{attribute 'linkalways'} 
{attribute 'no_explicit_call' := 'This FB is a CLASS and must be accessed using methods or properties'}
{attribute 'enable_dynamic_creation'}
FUNCTION_BLOCK ChunkableServerResponse IMPLEMENTS I_ServerResponse
VAR
	serverResponse : I_ServerResponse;
	chunkedResponseManager : I_ChunkedResponseManager;
END_VAR

METHOD PUBLIC Accepted
VAR_INPUT
END_VAR
serverResponse.Accepted();
END_METHOD

METHOD PUBLIC Busy
VAR_INPUT
END_VAR
serverResponse.Busy();
END_METHOD

METHOD PUBLIC Error
VAR_INPUT
	Message : T_MAXSTRING;
END_VAR
serverResponse.Error(Message);
END_METHOD

METHOD FB_init : BOOL
VAR_INPUT
	bInitRetains : BOOL; // if TRUE, the retain variables are initialized (warm start / cold start)
	bInCopyCode : BOOL;  // if TRUE, the instance afterwards gets moved into the copy code (online change)
	ServerResponse : I_ServerResponse;
	ChunkedResponseManager : I_ChunkedResponseManager;
END_VAR
THIS^.serverResponse := ServerResponse;
This^.chunkedResponseManager := ChunkedResponseManager;
END_METHOD

PROPERTY PUBLIC Header : I_ServerResponseHeader
GET
Header := serverResponse.Header;
END_GET
END_PROPERTY

PROPERTY PUBLIC HeadersSent : BOOL
GET
HeadersSent := serverResponse.HeadersSent;
END_GET
END_PROPERTY

METHOD PUBLIC Pending
VAR_INPUT
	ResponseId : T_MAXSTRING;
	RetryDelayInMs : UDINT;
END_VAR
serverResponse.Pending(ResponseId, RetryDelayInMs);
END_METHOD

METHOD PUBLIC Success
VAR_INPUT
	PayloadDataAddress : PVOID;
	PayloadDataSize : UDINT;
END_VAR
chunkedResponseManager.HandleSuccess(serverResponse, PayloadDataAddress, PayloadDataSize);
END_METHOD

END_FUNCTION_BLOCK

(* stored: Version 1.1.0.1, ProductVersion 3.1.4024.12
   POU ChunkableServerResponse: Id {1f49da79-fc35-4c8f-8220-dbaca20491ac}, SpecialFunc None
   Folder Constructor: Id {1ca7b83f-10b7-4590-a248-a044744ee4f1}
   Method Accepted: Id {b6d0e7df-fe49-4f21-af57-ccd2f060058f}
   Method Busy: Id {3b955f13-968e-4ac1-978c-3d20a4e8637e}
   Method Error: Id {f9d27d9c-8ba1-40c8-972d-c24b136a8e4b}
   Method FB_init: Id {5322a03e-2e39-4a02-a321-599436055475}
   Property Header: Id {1daa3846-b6e0-490b-bc19-d32f5a3f29c3}
   Get Get: Id {e5d490d6-a712-4f8e-b259-d2aac6a82b77}
   Property HeadersSent: Id {76d5ed19-c44f-48dc-9f9c-a6c85ef0aa6b}
   Get Get: Id {8be4dc39-b712-4ac0-b614-4bb76382010e}
   Method Pending: Id {e682f307-3e49-4896-95ea-6f74ef047fe7}
   Method Success: Id {900688fe-0167-4eee-bf11-e332ca2b544d} *)
